# B&R Automation Studio project mappViewGettingStarted1
Automation Studio 4.2.7.54 SP; technology packages: mappView 1.1.1

## Configuration Config1

CPU PC_any, AutomationRuntime J4.25, Build 4.1.2, Vc V4.25.0

### Task classes (Cpu.sw)
```
Cyclic#1 (cycle 100000 us, tolerance 10000000 us):
  Program <- Program.prg
Binaries: TCData, arconfig, asfw, ashwd, iomap, User, Role, sysconf
Libraries: MTBasics, brsystem, MTTypes, sys_lib, runtime, astime, asieccon
```

### Hardware
```
PC : PC_any v1.1.0.0 (OrderNumber=PC)
  ConfigurationID = mappViewGettingStarted_Config1
  Cyclic1Duration = 100000
  Cyclic1Tolerance = 10000000
  Cyclic2Duration = 200000
  Cyclic2Tolerance = 10000000
  Cyclic3Duration = 500000
  Cyclic3Tolerance = 10000000
  Cyclic4Duration = 1000000
  Cyclic4Tolerance = 10000000
  Cyclic5Duration = 2000000
  Cyclic5Tolerance = 10000000
  Cyclic6Duration = 3000000
  Cyclic6Tolerance = 12000000
  Cyclic7Duration = 4000000
  Cyclic7Tolerance = 12000000
  Cyclic8Duration = 5000000
  Cyclic8Tolerance = 30000000
  ActivateOpcUa = 1
  OpcUa_Security_SoftwareCertificates = 
  OpcUa_Security_AdminRole = Administrators
```

## Logical view

Binary libraries used (declarations not repeated): operator, runtime, astime, AsIecCon, MTBasics 2.20.0, brsystem, MTTypes 1.03.0, sys_lib

### Global.var - Global variables
```iecst
VAR
	SetTemperature : INT;
	CurrentTemperature : INT;
END_VAR
```


### Program Logical/Program (IEC)

#### Main.st - Init, cyclic, exit code
```iecst
PROGRAM _INIT
	SetTemperature := 35;
END_PROGRAM

PROGRAM _CYCLIC
	(*
		Using FUNCTION block MTBasicsPT1() TO
		implement a 1st order delay element (PT1).
	*)
	MTBasicsPT1_0.Enable := 1;
	MTBasicsPT1_0.Gain := 1;
	MTBasicsPT1_0.TimeConstant := 1;
	MTBasicsPT1_0.In := INT_TO_REAL(SetTemperature);

	MTBasicsPT1_0();

	CurrentTemperature := REAL_TO_INT(MTBasicsPT1_0.Out);

	(*
		generate saw tooth signal for further usage of TM641 exercises

	*)
	aiTankLevel := aiTankLevel + 1;

END_PROGRAM
```

#### Variables.var - Local variables
```iecst
VAR
	MTBasicsPT1_0 : MTBasicsPT1;
	aiTankLevel : USINT;
END_VAR
```

- Visualisation Logical/mappView (not shown)

Listed in the project but not available here: Logical/Global.typ
